(* 2. EMERGENCY STOP LOGIC (Error 12) *)
IF E_Stop_Active THEN
    FOR i := 1 TO 6 DO
        Auto_Bin[i] := FALSE;
        auto_bin_cutoff[i] := FALSE;
        auto_bin_motor[i] := FALSE;
    END_FOR;
    Sequence_Complete := FALSE;
    Active_Material_ID := 0;
    Active_Bin_ID := 0;
    Active_Target_Weight := 0.0;
    Error_Code := 12;
    Status_Message := 'Error 12: Emergency Stop Active!';
    Step := 99;
    Transition_Timer(IN := FALSE);
    Completion_Timer(IN := FALSE);
    RETURN;
END_IF;


(* 3. RECIPE SEQUENCE START *)
IF Step = 0 AND Start_Button THEN
    Step := 1;
    bin_last_weight := load_cell_value;
    Sequence_Complete := FALSE;
    Error_Code := 0;
    Status_Message := 'Auto Batch Started';
    Active_Target_Weight := 0.0;
    (* Clear actual weights and outputs on start *)
    FOR i := 1 TO 6 DO
        Actual_Weights[i] := 0.0;
        Auto_Bin[i] := FALSE;
        auto_bin_cutoff[i] := FALSE;
        auto_bin_motor[i] := FALSE;
    END_FOR;
END_IF;


(* 4. SEQUENCE CONTROL STATE MACHINE *)
CASE Step OF
    0:
        Active_Material_ID := 0;
        Active_Bin_ID := 0;
        Active_Target_Weight := 0.0;
        IF Error_Code = 0 THEN Status_Message := 'Auto Idle'; END_IF;
        
    1..6: (* Discharging Silos 1 to 6 *)
        Mat_Idx := Auto_Bin_Material_Mapping[Step];
        
        IF Mat_Idx = 0 THEN
            (* Skip this bin instantly *)
            Step := Step + 1;
        ELSE
            (* Fetch target weight from global Recipe_Weights array *)
            bin_set_value := GVL.Recipe_Weights[Mat_Idx];
            
            (* Calculate effective target weight (Looked up Target - Tolerance) *)
            target_act_bin := bin_set_value - Auto_Bin_Tolerance[Step];
            Active_Target_Weight := target_act_bin;
            
            (* Calculate weight added by current active bin *)
            actual_bin := load_cell_value - bin_last_weight;
            Actual_Weights[Step] := actual_bin;
            
            (* Calculate cutoff trigger threshold *)
            cutoff_trigger_weight := target_act_bin - Auto_Bin_Cutoff_Weights[Step];
            
            Active_Material_ID := Mat_Idx;
            Active_Bin_ID := Step;
            Status_Message := 'Auto Pouring';
            
            (* COARSE/FINE FEED TRANSITIONS WITH TOLERANCE OFFSETS *)
            IF actual_bin < cutoff_trigger_weight THEN
                (* Phase 1: Coarse Feed (Conveyor Motor ON, Main Valve ON, Fine Cutoff OFF) *)
                Auto_Bin[Step] := TRUE;
                auto_bin_cutoff[Step] := FALSE;
                auto_bin_motor[Step] := TRUE;
            ELSIF actual_bin < target_act_bin THEN
                (* Phase 2: Fine Feed (Conveyor Motor ON, Main Valve OFF, Fine Cutoff ON) *)
                Auto_Bin[Step] := FALSE;
                auto_bin_cutoff[Step] := TRUE;
                auto_bin_motor[Step] := TRUE;
            ELSE
                (* Phase 3: Completed (All OFF) *)
                Auto_Bin[Step] := FALSE;
                auto_bin_cutoff[Step] := FALSE;
                auto_bin_motor[Step] := FALSE;
                bin_last_weight := load_cell_value;
                Active_Target_Weight := 0.0;
                Step := 10 + Step; // Offset to separate transition states
            END_IF;
            
            (* RUNTIME CHECKS *)
            (* Check 21 & 22: Scale Limits *)
            IF load_cell_value > 500.0 THEN
                Error_Code := 21;
                Status_Message := 'Error 21: Scale Overloaded!';
                Step := 99;
                RETURN;
            ELSIF load_cell_value < 0.0 THEN
                Error_Code := 22;
                Status_Message := 'Error 22: Scale Underloaded/Fault!';
                Step := 99;
                RETURN;
            END_IF;
        END_IF;

    11..15: (* Transition Delays (Between Bins) *)
        Active_Material_ID := 0;
        Active_Bin_ID := 0;
        Active_Target_Weight := 0.0;
        Status_Message := 'Transition Delay';
        
        Transition_Timer(IN := TRUE, PT := Step_Delay_Time);
        IF Transition_Timer.Q THEN
            Transition_Timer(IN := FALSE);
            Step := (Step - 10) + 1; // Advance to next bin
        END_IF;
        
    16: (* Transition Delay After Last Bin (Bin 6) Closes *)
        Active_Material_ID := 0;
        Active_Bin_ID := 0;
        Active_Target_Weight := 0.0;
        Status_Message := 'Settling Last Bin';
        
        Transition_Timer(IN := TRUE, PT := Step_Delay_Time);
        IF Transition_Timer.Q THEN
            Transition_Timer(IN := FALSE);
            Step := 7; // Go to post-discharge wait step
        END_IF;

    7: (* Wait 2 Seconds After Closing the Last Bin *)
        Active_Material_ID := 0;
        Active_Bin_ID := 0;
        Active_Target_Weight := 0.0;
        Status_Message := 'Settling Delay';
        Completion_Timer(IN := TRUE, PT := Post_Complete_Delay);
        IF Completion_Timer.Q THEN
            Completion_Timer(IN := FALSE);
            Step := 8; // Proceed to reset last weight
        END_IF;
        
    8: (* Reset bin_last_weight to 0 & Complete *)
        Active_Material_ID := 0;
        Active_Bin_ID := 0;
        Active_Target_Weight := 0.0;
        Status_Message := 'Sequence Completed';
        bin_last_weight := 0.0;
        Sequence_Complete := TRUE;
        
        IF NOT Start_Button THEN
            Step := 0;
            Sequence_Complete := FALSE;
            (* Reset all actual weights at completion once start is released *)
            FOR i := 1 TO 6 DO
                Actual_Weights[i] := 0.0;
            END_FOR;
        END_IF;
        
    99: (* Error Abort state *)
        FOR i := 1 TO 6 DO 
            Auto_Bin[i] := FALSE; 
            auto_bin_cutoff[i] := FALSE;
            auto_bin_motor[i] := FALSE;
        END_FOR;
        Active_Material_ID := 0;
        Active_Bin_ID := 0;
        Active_Target_Weight := 0.0;
        IF NOT Start_Button THEN
            Step := 0;
            Error_Code := 0;
            Status_Message := 'Auto Idle';
        END_IF;
END_CASE;

END_FUNCTION_BLOCK

// PLC_AC500_V3/Application/Manual_Batching_V9
FUNCTION_BLOCK Manual_Batching_V9
VAR_INPUT
    Start_Button : BOOL;      // Signal to start the batching sequence
    E_Stop_Active : BOOL;     // Emergency Stop active signal
    Manual_Bin_Material_Mapping : ARRAY[1..10] OF INT; // Material index mapping for 10 manual silos
    Manual_Bin_Cutoff_Weights : ARRAY[1..10] OF REAL; // Cutoff weight thresholds (kg)
    Manual_Bin_Tolerance : ARRAY[1..10] OF REAL; // Tolerance weight offset values (kg)
END_VAR
VAR_IN_OUT
    load_cell_value : REAL;   // Weight value read/written from load cell
END_VAR
VAR_OUTPUT
    Manual_Bin : ARRAY[1..10] OF BOOL; // Prompts/indicators for Bins 7..16
    manual_bin_cutoff : ARRAY[1..10] OF BOOL; // Manual pre-cutoff indicators
    manual_bin_motor : ARRAY[1..10] OF BOOL; // Main manual feeder motor outputs
    Actual_Weights : ARRAY[1..10] OF REAL; // Actual weight poured per silo
    Sequence_Complete : BOOL;  // Batch complete flag
    Active_Material_ID : INT;  // Currently active ingredient ID
    Active_Bin_ID : INT;       // Currently active physical Bin ID (7..16)
    Active_Target_Weight : REAL; // Recipe target weight of active bin (with tolerance applied)
    Error_Code : INT;          // Active error code
    Status_Message : STRING;   // Diagnostic text message
END_VAR
VAR
    Step : INT := 0;          // State machine index (0: Idle, 1..10: Bins, 11..20: Delays, 30: Settling, 40: Complete, 99: Error)
    bin_last_weight : REAL;   // Baseline weight on the load cell before starting current bin
    actual_bin : REAL;        // Current weight added from active bin
    target_act_bin : REAL;    // Effective target weight to add from the active bin (GVL target - Tolerance)
    bin_set_value : REAL;     // Setpoint weight looked up from GVL
    cutoff_trigger_weight : REAL; // Calculated target threshold weight minus cutoff and tolerance values
    
    Mat_Idx : INT;
    i : INT;                  // General loop index
    
    (* TIMERS FOR TRANSITIONS & DELAYS *)
    Transition_Timer : TON;
    Completion_Timer : TON;
    Step_Delay_Time : TIME := T#2S;
    Post_Complete_Delay : TIME := T#2S;
    
    (* DIAGNOSTIC TIMERS *)
    Operator_Timer : TON;
    
    (* SELF-CONTAINED SIMULATION VARIABLES *)
    Simulation_Mode : BOOL := TRUE;
    Sim_Rate : REAL := 10.0;            // Simulated pouring speed (10.0 kg/s)
    Sim_Timer : TON;
    Start_Sim_Weight : REAL;
    Discharge_Active : BOOL;
END_VAR

(* Manual Batching FB V9 with Tolerance Logic *)

(* 1. SIMULATION WEIGHT MANAGEMENT *)
IF Simulation_Mode AND Step <> 99 THEN
    (* Reset simulation to baseline *)
    IF Step = 0 AND NOT Start_Button AND NOT Sequence_Complete THEN
        load_cell_value := 0.0;
        bin_last_weight := 0.0;
        Start_Sim_Weight := 0.0;
        Sim_Timer(IN := FALSE);
    END_IF;
    
    (* Check if operator is actively pouring *)
    Discharge_Active := FALSE;
    IF Step >= 1 AND Step <= 10 THEN
        Discharge_Active := manual_bin_motor[Step];
    END_IF;
    
    (* Simulate weight gain on the load cell *)
    IF Discharge_Active THEN
        Sim_Timer(IN := TRUE, PT := T#1000S);
        load_cell_value := Start_Sim_Weight + (TIME_TO_REAL(Sim_Timer.ET) / 1000.0) * Sim_Rate;
    ELSE
        Sim_Timer(IN := FALSE);
        Start_Sim_Weight := load_cell_value;
    END_IF;
END_IF;


(* 2. EMERGENCY STOP LOGIC (Error 12) *)
IF E_Stop_Active THEN
    FOR i := 1 TO 10 DO
        Manual_Bin[i] := FALSE;
        manual_bin_cutoff[i] := FALSE;
        manual_bin_motor[i] := FALSE;
    END_FOR;
    Sequence_Complete := FALSE;
    Active_Material_ID := 0;
    Active_Bin_ID := 0;
    Active_Target_Weight := 0.0;
    Error_Code := 12;
    Status_Message := 'Error 12: Emergency Stop Active!';
    Step := 99;
    Transition_Timer(IN := FALSE);
    Completion_Timer(IN := FALSE);
    RETURN;
END_IF;


(* 3. RECIPE SEQUENCE START *)
IF Step = 0 AND Start_Button THEN
    Step := 1;
    bin_last_weight := load_cell_value;
    Sequence_Complete := FALSE;
    Error_Code := 0;
    Status_Message := 'Manual Batch Started';
    Active_Target_Weight := 0.0;
    (* Clear actual weights on start *)
    FOR i := 1 TO 10 DO
        Actual_Weights[i] := 0.0;
        Manual_Bin[i] := FALSE;
        manual_bin_cutoff[i] := FALSE;
        manual_bin_motor[i] := FALSE;
    END_FOR;
END_IF;


(* 4. SEQUENCE CONTROL STATE MACHINE *)
CASE Step OF
    0:
        Active_Material_ID := 0;
        Active_Bin_ID := 0;
        Active_Target_Weight := 0.0;
        IF Error_Code = 0 THEN Status_Message := 'Manual Idle'; END_IF;
        
    1..10: (* Prompts Silos 7 to 16 *)
        Mat_Idx := Manual_Bin_Material_Mapping[Step];
        
        IF Mat_Idx = 0 THEN
            (* Skip this bin instantly *)
            Step := Step + 1;
        ELSE
            (* Fetch target weight from global Recipe_Weights array *)
            bin_set_value := GVL.Recipe_Weights[Mat_Idx];
            
            (* Calculate effective target weight (Looked up Target - Tolerance) *)
            target_act_bin := bin_set_value - Manual_Bin_Tolerance[Step];
            Active_Target_Weight := target_act_bin;
            
            (* Calculate weight added by current active bin *)
            actual_bin := load_cell_value - bin_last_weight;
            Actual_Weights[Step] := actual_bin;
            
            (* Calculate cutoff trigger threshold *)
            cutoff_trigger_weight := target_act_bin - Manual_Bin_Cutoff_Weights[Step];
            
            Active_Material_ID := Mat_Idx;
            Active_Bin_ID := Step + 6;
            Status_Message := 'Manual Pouring Active';
            
            (* COARSE/FINE FEED TRANSITIONS WITH TOLERANCE OFFSETS *)
            IF actual_bin < cutoff_trigger_weight THEN
                (* Phase 1: Coarse Feed (Motor ON, Prompt ON, Cutoff OFF) *)
                Manual_Bin[Step] := TRUE;
                manual_bin_cutoff[Step] := FALSE;
                manual_bin_motor[Step] := TRUE;
            ELSIF actual_bin < target_act_bin THEN
                (* Phase 2: Fine Feed (Motor ON, Prompt OFF, Cutoff ON) *)
                Manual_Bin[Step] := FALSE;
                manual_bin_cutoff[Step] := TRUE;
                manual_bin_motor[Step] := TRUE;
            ELSE
                (* Phase 3: Completed (All OFF) *)
                Manual_Bin[Step] := FALSE;
                manual_bin_cutoff[Step] := FALSE;
                manual_bin_motor[Step] := FALSE;
                bin_last_weight := load_cell_value;
                Active_Target_Weight := 0.0;
                Step := 10 + Step; // Offset to separate transition states
            END_IF;
            
            (* RUNTIME CHECKS *)
            (* Check 21 & 22: Scale Limits *)
            IF load_cell_value > 500.0 THEN
                Error_Code := 21;
                Status_Message := 'Error 21: Scale Overloaded!';
                Step := 99;
                RETURN;
            ELSIF load_cell_value < 0.0 THEN
                Error_Code := 22;
                Status_Message := 'Error 22: Scale Underloaded/Fault!';
                Step := 99;
                RETURN;
            END_IF;
            
            (* Check 30: Operator Timeout *)
            Operator_Timer(IN := manual_bin_motor[Step], PT := T#300S);
            IF Operator_Timer.Q THEN
                Error_Code := 30;
                Status_Message := 'Error 30: Manual Operator Timeout!';
                Step := 99;
                RETURN;
            END_IF;
        END_IF;

    11..19: (* Transition Delays (Between Bins) *)
        Active_Material_ID := 0;
        Active_Bin_ID := 0;
        Active_Target_Weight := 0.0;
        Status_Message := 'Transition Delay';
        Transition_Timer(IN := TRUE, PT := Step_Delay_Time);
        IF Transition_Timer.Q THEN
            Transition_Timer(IN := FALSE);
            Step := (Step - 10) + 1; // Advance to next bin
        END_IF;
        
    20: (* Transition Delay After Last Bin (Bin 10) Closes *)
        Active_Material_ID := 0;
        Active_Bin_ID := 0;
        Active_Target_Weight := 0.0;
        Status_Message := 'Settling Last Bin';
        Transition_Timer(IN := TRUE, PT := Step_Delay_Time);
        IF Transition_Timer.Q THEN
            Transition_Timer(IN := FALSE);
            Step := 30; // Go to post-discharge wait step (State 30)
        END_IF;

    30: (* Wait 2 Seconds After Closing the Last Bin *)
        Active_Material_ID := 0;
        Active_Bin_ID := 0;
        Active_Target_Weight := 0.0;
        Status_Message := 'Settling Delay';
        Completion_Timer(IN := TRUE, PT := Post_Complete_Delay);
        IF Completion_Timer.Q THEN
            Completion_Timer(IN := FALSE);
            Step := 40; // Proceed to reset last weight (State 40)
        END_IF;
        
    40: (* Reset bin_last_weight to 0 & Complete *)
        Active_Material_ID := 0;
        Active_Bin_ID := 0;
        Active_Target_Weight := 0.0;
        Status_Message := 'Sequence Completed';
        bin_last_weight := 0.0;
        Sequence_Complete := TRUE;
        
        IF NOT Start_Button THEN
            Step := 0;
            Sequence_Complete := FALSE;
            (* Reset all actual weights at completion once start is released *)
            FOR i := 1 TO 10 DO
                Actual_Weights[i] := 0.0;
            END_FOR;
        END_IF;
        
    99: (* Error Abort state *)
        FOR i := 1 TO 10 DO 
            Manual_Bin[i] := FALSE;
            manual_bin_cutoff[i] := FALSE;
            manual_bin_motor[i] := FALSE;
        END_FOR;
        Active_Material_ID := 0;
        Active_Bin_ID := 0;
        Active_Target_Weight := 0.0;
        IF NOT Start_Button THEN
            Step := 0;
            Error_Code := 0;
            Status_Message := 'Manual Idle';
        END_IF;
END_CASE;

END_FUNCTION_BLOCK

// PLC_AC500_V3/Application/batching9
PROGRAM batching9
VAR
    Auto_Ctrl : Auto_Batching_V9;
    Manual_Ctrl : Manual_Batching_V9;
    
    (* Global Inputs & Toggles *)
    Start_Button : BOOL;
    E_Stop_Active : BOOL;
    
    (* Parallel Weight Feedbacks *)
    load_cell_auto : REAL;
    load_cell_manual : REAL;
    
    (* Sub-Block Diagnostic Indicators - Ordered exactly below loadcell *)
    Auto_Active_Mat : INT;
    Auto_Active_Bin : INT;
    Auto_Active_Target : REAL; // Active Target Weight for Auto (displays GVL setpoint - Tolerance)
    Auto_Err : INT;
    Auto_Msg : STRING;
    
    Manual_Active_Mat : INT;
    Manual_Active_Bin : INT;
    Manual_Active_Target : REAL; // Active Target Weight for Manual (displays GVL setpoint - Tolerance)
    Manual_Err : INT;
    Manual_Msg : STRING;
    
    (* Process Outputs *)
    Auto_Bin : ARRAY[1..6] OF BOOL; // Valve control outputs (Coarse)
    auto_bin_cutoff : ARRAY[1..6] OF BOOL; // Cutoff indicators (Fine)
    auto_bin_motor : ARRAY[1..6] OF BOOL; // Conveyor/feeder motor outputs
    
    Manual_Bin : ARRAY[1..10] OF BOOL; // Prompt indicators (Coarse)
    manual_bin_cutoff : ARRAY[1..10] OF BOOL; // Cutoff indicators (Fine)
    manual_bin_motor : ARRAY[1..10] OF BOOL; // Conveyor/feeder motor outputs
    
    Auto_Weights : ARRAY[1..6] OF REAL;
    Manual_Weights : ARRAY[1..10] OF REAL;
    
    Auto_Complete : BOOL;
    Manual_Complete : BOOL;
    Sequence_Complete : BOOL;
    
    (* Diagnostics & Interlocks *)
    Error_Code : INT := 0;
    Status_Message : STRING := 'System Ready';
    
    (* Array Configurations & Mapping - Renamed for clarity *)
    Auto_Bin_Material_Mapping : ARRAY[1..6] OF INT := [1, 2, 0, 4, 5, 6];
    Manual_Bin_Material_Mapping : ARRAY[1..10] OF INT := [7, 8, 0, 10, 11, 12, 13, 14, 15, 16];
    Auto_Bin_Cutoff_Weights : ARRAY[1..6] OF REAL := [2.0, 1.5, 0.0, 3.0, 5.0, 1.0]; // Cutoff margins (kg)
    Manual_Bin_Cutoff_Weights : ARRAY[1..10] OF REAL := [2.0, 1.5, 0.0, 3.0, 5.0, 1.0, 2.0, 2.0, 2.0, 2.0];
    Auto_Bin_Tolerance : ARRAY[1..6] OF REAL := [1.0, 0.5, 0.0, 1.0, 2.0, 0.5]; // Tolerance offsets (kg)
    Manual_Bin_Tolerance : ARRAY[1..10] OF REAL := [1.0, 0.5, 0.0, 1.0, 2.0, 0.5, 1.0, 1.0, 1.0, 1.0];
    
    i : INT;
    j : INT;
    Duplicate_Found : BOOL;
    Invalid_Material_Range : BOOL;
    Zero_Target_Found : BOOL;
    Conf_Err_Id : INT;
END_VAR

(* 1. STARTUP CONFIGURATION CHECKS *)
Duplicate_Found := FALSE;
Invalid_Material_Range := FALSE;
Zero_Target_Found := FALSE;

FOR i := 1 TO 6 DO
    (* Check 2: Out of Range (Auto) *)
    IF Auto_Bin_Material_Mapping[i] < 0 OR Auto_Bin_Material_Mapping[i] > 20 THEN
        Invalid_Material_Range := TRUE;
    END_IF;
    
    (* Check 3: Zero Target (Auto) *)
    IF Auto_Bin_Material_Mapping[i] <> 0 AND Auto_Bin_Material_Mapping[i] <= 20 THEN
        IF GVL.Recipe_Weights[Auto_Bin_Material_Mapping[i]] = 0.0 THEN
            Zero_Target_Found := TRUE;
        END_IF;
    END_IF;
    
    (* Check 1: Duplicate Cross-Array Material ID *)
    IF Auto_Bin_Material_Mapping[i] <> 0 AND Auto_Bin_Material_Mapping[i] <= 20 THEN
        FOR j := 1 TO 10 DO
            IF Auto_Bin_Material_Mapping[i] = Manual_Bin_Material_Mapping[j] THEN
                Duplicate_Found := TRUE;
            END_IF;
        END_FOR;
    END_IF;
END_FOR;

FOR j := 1 TO 10 DO
    (* Check 2: Out of Range (Manual) *)
    IF Manual_Bin_Material_Mapping[j] < 0 OR Manual_Bin_Material_Mapping[j] > 20 THEN
        Invalid_Material_Range := TRUE;
    END_IF;
    
    (* Check 3: Zero Target (Manual) *)
    IF Manual_Bin_Material_Mapping[j] <> 0 AND Manual_Bin_Material_Mapping[j] <= 20 THEN
        IF GVL.Recipe_Weights[Manual_Bin_Material_Mapping[j]] = 0.0 THEN
            Zero_Target_Found := TRUE;
        END_IF;
    END_IF;
END_FOR;

(* Configuration Error Resolution *)
IF Duplicate_Found THEN
    Error_Code := 1;
    Status_Message := 'Error 1: Duplicate Material ID mapped in Auto and Manual!';
ELSIF Invalid_Material_Range THEN
    Error_Code := 2;
    Status_Message := 'Error 2: Material Index configuration out of range (1..20)!';
ELSIF Zero_Target_Found THEN
    Error_Code := 3;
    Status_Message := 'Error 3: Configured Material ID has a 0.0 kg target weight!';
ELSE
    IF Error_Code <= 3 THEN
        Error_Code := 0;
    END_IF;
END_IF;

(* Abort sequences if a configuration error exists *)
IF Error_Code >= 1 AND Error_Code <= 3 THEN
    FOR i := 1 TO 6 DO Auto_Bin[i] := FALSE; auto_bin_cutoff[i] := FALSE; auto_bin_motor[i] := FALSE; END_FOR;
    FOR i := 1 TO 10 DO Manual_Bin[i] := FALSE; manual_bin_cutoff[i] := FALSE; manual_bin_motor[i] := FALSE; END_FOR;
    Auto_Ctrl(Start_Button := FALSE, E_Stop_Active := TRUE, load_cell_value := load_cell_auto);
    Manual_Ctrl(Start_Button := FALSE, E_Stop_Active := TRUE, load_cell_value := load_cell_manual);
    Auto_Active_Target := 0.0;
    Manual_Active_Target := 0.0;
    RETURN;
END_IF;


(* 2. CONCURRENT EXECUTION OF FB INSTANCES *)
Auto_Ctrl(
    Start_Button := Start_Button,
    E_Stop_Active := E_Stop_Active,
    load_cell_value := load_cell_auto,
    Auto_Bin_Material_Mapping := Auto_Bin_Material_Mapping,
    Auto_Bin_Cutoff_Weights := Auto_Bin_Cutoff_Weights,
    Auto_Bin_Tolerance := Auto_Bin_Tolerance,
    Auto_Bin => Auto_Bin,
    auto_bin_cutoff => auto_bin_cutoff,
    auto_bin_motor => auto_bin_motor,
    Actual_Weights => Auto_Weights,
    Sequence_Complete => Auto_Complete,
    Active_Material_ID => Auto_Active_Mat,
    Active_Bin_ID => Auto_Active_Bin,
    Active_Target_Weight => Auto_Active_Target,
    Error_Code => Auto_Err,
    Status_Message => Auto_Msg
);

Manual_Ctrl(
    Start_Button := Start_Button,
    E_Stop_Active := E_Stop_Active,
    load_cell_value := load_cell_manual,
    Manual_Bin_Material_Mapping := Manual_Bin_Material_Mapping,
    Manual_Bin_Cutoff_Weights := Manual_Bin_Cutoff_Weights,
    Manual_Bin_Tolerance := Manual_Bin_Tolerance,
    Manual_Bin => Manual_Bin,
    manual_bin_cutoff => manual_bin_cutoff,
    manual_bin_motor => manual_bin_motor,
    Actual_Weights => Manual_Weights,
    Sequence_Complete => Manual_Complete,
    Active_Material_ID => Manual_Active_Mat,
    Active_Bin_ID => Manual_Active_Bin,
    Active_Target_Weight => Manual_Active_Target,
    Error_Code => Manual_Err,
    Status_Message => Manual_Msg
);

(* Runtime Error Mapping & Aggregation *)
IF Auto_Err <> 0 THEN
    Error_Code := Auto_Err;
    Status_Message := CONCAT('Auto Error: ', Auto_Msg);
ELSIF Manual_Err <> 0 THEN
    Error_Code := Manual_Err;
    Status_Message := CONCAT('Manual Error: ', Manual_Msg);
ELSE
    Error_Code := 0;
    
    Sequence_Complete := Auto_Complete AND Manual_Complete;
    IF Sequence_Complete THEN
        Status_Message := 'Batch Sequence Completed';
    ELSIF Start_Button THEN
        Status_Message := 'Batch Sequence Running';
    ELSE
        Status_Message := 'System Ready';
    END_IF;
END_IF;

END_PROGRAM

// PLC_AC500_V3/Application/batching4_vis
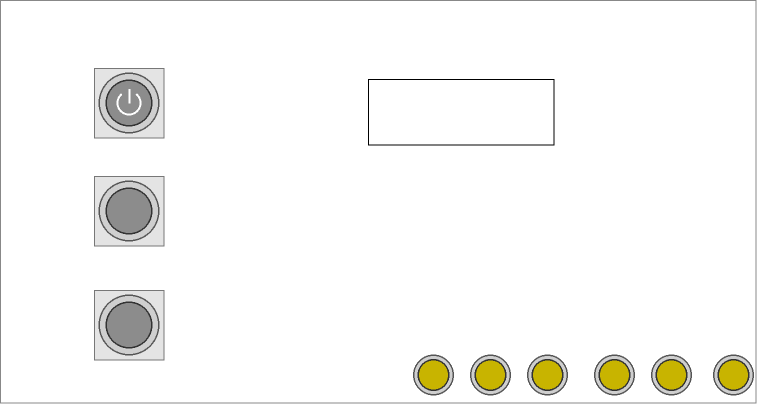
VISUALIZATION batching4_vis  // 757x404
    PushSwitch (94,290 70x70), behaviour: TOGGLE, style: Switch-PushSwitch-Gray
    PushSwitch (94,176 70x70), behaviour: TOGGLE, style: Switch-PushSwitch-Gray
    PowerSwitch (94,68 70x70), behaviour: TOGGLE, style: Switch-PowerSwitch-Gray
    Lamp1 (591,346 47x58), style: Lamp-Lamp1-Yellow
    Lamp1 (524,346 47x58), style: Lamp-Lamp1-Yellow
    Lamp1 (467,346 47x58), style: Lamp-Lamp1-Yellow
    Lamp1 (410,346 47x58), style: Lamp-Lamp1-Yellow
    Lamp1 (648,346 47x58), style: Lamp-Lamp1-Yellow
    Lamp1 (710,346 47x58), style: Lamp-Lamp1-Yellow
    Rectangle (368,79 186x66)
END_VISUALIZATION

(* text list Diag_IO_Bus (id | default | en | de | fr | es | zh)
  Err_1037 | Test error | Test error | Testfehler |  |  | 测试错误
  Err_12 | Test pulse error -> Check wiring and sensor | Test pulse error -> Check wiring and sensor | Testimpuls-Fehler -> Verdrahtung und Sensor prüfen |  |  | 测试脉冲错误 -> 检查接线和传感器
  Err_13 | Test pulse cross-talk error -> Check wiring and sensor. If this error persists, replace I/O module. Contact ABB technical support. | Test pulse cross-talk error -> Check wiring and sensor. If this error persists, replace I/O module. Contact ABB technical support. | Fehler Testimpuls Kanalübersprechen  -> Verdrahtung und Sensor prüfen. Falls der Fehler weiterhin besteht, E/A-Modul austauschen. Technischen Support von ABB kontaktieren. |  |  | 测试脉冲串扰错误 -> 检查接线和传感器. 如果此错误仍然存在，请更换 I/O 模块. 联系 ABB 技术支持.
  Err_16128 | Failed max wait run | Failed max wait run | Lauf max. Warten fehlgeschlagen |  |  | 最大等待运行失败
  Err_16129 | Critical error, see log | Critical error, see log | Kritischer Fehler, siehe Protokoll |  |  | 严重错误，请参阅日志
  Err_16130 | Fatal error, see log | Fatal error, see log | Schwerwiegender Fehler, siehe Protokoll |  |  | 致命错误，请参阅日志
  Err_16131 | Timeout -> Replace I/O module | Timeout -> Replace I/O module | Timeout -> E/A-Modul austauschen |  |  | 超时 -> 更换 I/O 模块
  Err_16133 | Output data size mismatch | Output data size mismatch | Diskrepanz Ausgangsdatengröße |  |  | 输出数据大小不匹配
  Err_16134 | Input data size mismatch | Input data size mismatch | Diskrepanz Eingangsdatengröße |  |  | 输入数据大小不匹配
  Err_16137 | Overflow diagnosis buffer -> Restart | Overflow diagnosis buffer -> Restart | Überlauf Diagnosepuffer -> Neu Starten |  |  | 诊断缓冲区溢出 -> 重新启动
  Err_16138 | Non-safety I/O: Voltage overflow at outputs (above UP3 level), Safety I/O: Process voltage too high -> Check terminals / Check process voltage | Non-safety I/O: Voltage overflow at outputs (above UP3 level), Safety I/O: Process voltage too high -> Check terminals / Check process voltage | Standard-E/A: Spannungsüberlauf an Ausgängen (über UP3-Niveau), Sicherheits-E/A: Prozessspannung zu hoch -> Terminals prüfen / Prozessspannung prüfen |  |  | 非安全 I/O：输出端电压溢出（高于 UP3 电平），安全 I/O：过程电压过高 -> 检查终端 / 检查过程电压
  Err_16139 | Process voltage UP or UP3 too low -> Check process voltage | Process voltage UP or UP3 too low -> Check process voltage | Prozessspannung UP oder UP3 zu niedrig -> Prozessspannung prüfen |  |  | 过程电压 UP 或 UP3 过低 -> 检查过程电压
  Err_16145 | Error setting parameters | Error setting parameters | Fehlereinstellungsparameter |  |  | 设置参数时出错
  Err_16146 | Plausibility check failed (iParameter) -> Check configuration | Plausibility check failed (iParameter) -> Check configuration | Plausibilitätsprüfung fehlgeschlagen (iParameter) -> Konfiguration überprüfen |  |  | 合理性检查失败（i 参数） -> 检查配置
  Err_16147 | Checksum error -> Non-safety I/O: Replace I/O module. Safety I/O: Check safety configuration and CRCs for I- and F-Parameters. | Checksum error -> Non-safety I/O: Replace I/O module. Safety I/O: Check safety configuration and CRCs for I- and F-Parameters. | Prüfsummenfehler -> Standard-E/A: E/A-Modul austauschen. Sicherheits-E/A: Sicherheitskonfiguration und CRCs auf I- und F-Parameter prüfen. |  |  | 检校验和错误 -> 非安全 I/O：更换 I/O 模块. 安全 I/O：检查 I 参数和 F 参数的安全配置和 CRC.
  Err_16148 | PROFIsafe communication error -> Restart I/O module. If this error persists, contact ABB technical support. | PROFIsafe communication error -> Restart I/O module. If this error persists, contact ABB technical support. | PROFIsafe-Kommunikationsfehler -> E/A-Modul neu starten. Falls der Fehler weiterhin besteht, technischen Support von ABB kontaktieren. |  |  | PROFIsafe 通信错误 -> 重新启动 I/O 模块. 如果此错误仍然存在，请联系 ABB 技术支持.
  Err_16149 | No module data | No module data | Keine Moduldaten |  |  | 无模块数据
  Err_16153 | PROFIsafe watchdog timed out -> Restart I/O module. If this error persists, increase PROFIsafe watchdog time. | PROFIsafe watchdog timed out -> Restart I/O module. If this error persists, increase PROFIsafe watchdog time. | Timeout von PROFIsafe-Watchdog -> E/A-Modul neu starten. Falls der Fehler weiterhin besteht, PROFIsafe-Watchdog-Zeit verlängern. |  |  | PROFIsafe 看门狗超时 -> 重新启动 I/O 模块. 如果此错误仍然存在，请增加 PROFIsafe 看门狗时间.
  Err_16154 | Size of parameters expected by module differs from size provided by configuration -> Check master or configuration | Size of parameters expected by module differs from size provided by configuration -> Check master or configuration | Vom Modul erwartete Parametergröße weicht von der in der Konfiguration angegebenen Größe ab -> Master oder Konfiguration überprüfen |  |  | 模块期望的参数大小与配置提供的参数大小不同 -> 检查主设备或配置
  Err_16156 | F-Parameter configuration and address switch value do not match -> Check I/O module F-Parameter configuration and module address switch value. | F-Parameter configuration and address switch value do not match -> Check I/O module F-Parameter configuration and module address switch value. | Konfiguration für F-Parameter und Wert des Adressschalters stimmen nicht überein -> Konfiguration für F-Parameter des E/A-Moduls und Wert des Adressschalters überprüfen. |  |  | F 参数配置和地址开关值不匹配 -> 检查 I/O 模块 F 参数配置和模块地址开关值.
  Err_16158 | Type of present module does not match configuration | Type of present module does not match configuration | Typ des vorhandenen Moduls stimmt nicht mit Konfiguration überein |  |  | 当前模块类型与配置不匹配
  Err_16159 | Configured number of modules differs from found ones | Configured number of modules differs from found ones | Konfigurierte Anzahl von Modulen weicht von Anzahl gefundener Module ab |  |  | 配置的模块数量与找到的模块数量不同
  Err_16160 | At least one module failed during configuration | At least one module failed during configuration | Mindestens ein Modul während Konfiguration ausgefallen |  |  | 配置期间至少有一个模块发生故障
  Err_16164 | Internal data exchange failure -> Replace I/O module | Internal data exchange failure -> Replace I/O module | Fehler interner Datenaustausch -> E/A-Modul austauschen |  |  | 内部数据交换失败 -> 更换 I/O 模块
  Err_16168 | Different hard-/firmware versions in the module -> Replace I/O module | Different hard-/firmware versions in the module -> Replace I/O module | Unterschiedliche Hardware-/Firmware-Versionen im Modul -> E/A-Modul austauschen |  |  | 模块中的硬件/固件版本不同 -> 更换 I/O 模块
  Err_16171 | Internal error -> Replace I/O module | Internal error -> Replace I/O module | Interner Fehler -> E/A-Modul austauschen |  |  | 内部错误 -> 更换 I/O 模块
  Err_16172 | Has not passed factory test | Has not passed factory test | Hat Werksprüfung nicht bestanden |  |  | 未通过出厂测试
  Err_16173 | No process voltage UP or UP3 -> Check process voltage | No process voltage UP or UP3 -> Check process voltage | Keine Prozessspannung UP oder UP3 -> Prozessspannung prüfen |  |  | 无过程电压 UP 或 UP3 -> 检查过程电压
  Err_16175 | Sensor voltage too low | Sensor voltage too low | Sensorspannung zu niedrig |  |  | 传感器电压过低
  Err_16194 | Fatal error, not running any more | Fatal error, not running any more | Schwerwiegender Fehler, Ausführung gestoppt |  |  | 致命错误，不再运行
  Err_16246 | Failed to start the parameterization of modules | Failed to start the parameterization of modules | Starten von Parametrierung für Module fehlgeschlagen |  |  | 无法启动模块的参数化
  Err_16247 | Failed setting parameters | Failed setting parameters | Einstellen von Parametern fehlgeschlagen |  |  | 设置参数失败
  Err_16248 | Failed setting expected module | Failed setting expected module | Einstellen des erwarteten Moduls fehlgeschlagen |  |  | 设置预期模块失败
  Err_16254 | Size of parameters expected by module differs from size provided by configuration | Size of parameters expected by module differs from size provided by configuration | Vom Modul erwartete Parametergröße weicht von der in der Konfiguration angegebenen Größe ab |  |  | 模块期望的参数大小与配置提供的参数大小不同
  Err_18 | Test error | Test error | Testfehler |  |  | 测试错误
  Err_25 | Stuck at error -> Check I/O module wiring. Restart I/O module, if needed. If this error persists, replace I/O module. | Stuck at error -> Check I/O module wiring. Restart I/O module, if needed. If this error persists, replace I/O module. | Hängengeblieben bei Fehler -> Verdrahtung des E/A-Moduls überprüfen. Bei Bedarf E/A-Modul neu starten. Falls der Fehler weiterhin besteht, E/A-Modul austauschen. |  |  | 卡在错误处 -> 检查 I/O 模块接线. 如果需要，重新启动 I/O 模块. 如果此错误仍然存在，请更换 I/O 模块.
  Err_257 | Wrong measurement, false temperature at the compensation channel | Wrong measurement, false temperature at the compensation channel | Falscher Messwert, falsche Temperatur an Kompensationskanal |  |  | 测量值错误，补偿通道温度错误
  Err_258 | AI531: Wrong measurement; potential difference is too high; CD522: PWM duty cycle out of duty area | AI531: Wrong measurement; potential difference is too high; CD522: PWM duty cycle out of duty area | AI531: Falscher Messwert; Potenzialdifferenz zu hoch; CD522: PWM-Einschaltdauer außerhalb des Einschaltbereichs |  |  | AI531：测量错误; 电位差过高; CD522: PWM 占空比超出占空比范围
  Err_260 | Measurement overflow -> Check channel wiring and sensor power supply | Measurement overflow -> Check channel wiring and sensor power supply | Messwertüberschreitung -> Kanalverdrahtung und Spannungsversorgung des Sensors prüfen |  |  | 测量值溢出 -> 检查通道接线和传感器电源
  Err_263 | Measurement underflow -> Check channel wiring and sensor power supply | Measurement underflow -> Check channel wiring and sensor power supply | Messwertunterschreitung -> Kanalverdrahtung und Spannungsversorgung des Sensors prüfen |  |  | 测量值下溢 -> 检查通道接线和传感器电源
  Err_266 | Short circuit and cut wire or "out of range" | Short circuit and cut wire or "out of range" | Kurzschluss und Drahtbruch oder „außerhalb des zulässigen Bereichs“ |  |  | 短路和断线或“超出范围”
  Err_267 | Output/process voltage too low | Output/process voltage too low | Ausgangs-/Prozessspannung zu gering |  |  | 输出/过程电压过低
  Err_273 | Test error | Test error | Testfehler |  |  | 测试错误
  Err_28 | Cross-talk error -> Check I/O module wiring. Restart I/O module, if needed. If this error persists, replace I/O module. | Cross-talk error -> Check I/O module wiring. Restart I/O module, if needed. If this error persists, replace I/O module. | Fehler Kanalübersprechen -> Verdrahtung des E/A-Moduls überprüfen. Bei Bedarf E/A-Modul neu starten. Falls der Fehler weiterhin besteht, E/A-Modul austauschen. |  |  | 串扰错误 -> 检查 I/O 模块接线. 如果需要，重新启动 I/O 模块. 如果此错误仍然存在，请更换 I/O 模块.
  Err_3 | Discrepancy time expired -> Check discrepancy time value, channel wiring and sensor. | Discrepancy time expired -> Check discrepancy time value, channel wiring and sensor. | Diskrepanzzeit abgelaufen -> Diskrepanzzeit-Wert, Kanalverdrahtung und Sensor überprüfen. |  |  | 偏差时间已过 -> 检查差异时间值、通道接线和传感器.
  Err_303 | Short circuit at analog input -> Check channel wiring | Short circuit at analog input -> Check channel wiring | Kurzschluss an Analogeingang -> Kanalverdrahtung prüfen |  |  | 模拟输入端短路 -> 检查通道接线
  Err_304 | Analog value overflow or broken wire at an analog input -> Check value or check terminals | Analog value overflow or broken wire at an analog input -> Check value or check terminals | Analogwert-Überlauf oder Drahtbruch an Analogeingang -> Wert oder Terminals prüfen |  |  | 模拟输入端模拟值溢出或断线 -> 检查值或检查终端
  Err_311 | Value difference too high -> Adjust tolerance window for channels. Check channel wiring and sensor configuration. | Value difference too high -> Adjust tolerance window for channels. Check channel wiring and sensor configuration. | Wertdifferenz zu groß -> Toleranzfenster für Kanäle einstellen. Kanalverdrahtung und Sensorkonfiguration prüfen. |  |  | 值差异过大 -> 调整通道的容差范围. 检查通道接线和传感器配置.
  Err_524 | Stuck at error | Stuck at error | Hängengeblieben bei Fehler |  |  | 卡在错误处
  Err_525 | Readback error -> Check I/O module wiring. Restart I/O module, if needed. If this error persists, replace I/O module. | Readback error -> Check I/O module wiring. Restart I/O module, if needed. If this error persists, replace I/O module. | Fehler Rücklesen -> Verdrahtung des E/A-Moduls überprüfen. Bei Bedarf E/A-Modul neu starten. Falls der Fehler weiterhin besteht, E/A-Modul austauschen. |  |  | 回读错误 -> 检查 I/O 模块接线. 如果需要，重新启动 I/O 模块. 如果此错误仍然存在，请更换 I/O 模块.
  Err_530 | Class 3: Cross-talk error; Class 4: Internal fuse at 0V is defect. 0V not connected with GND -> Check I/O module wiring. Restart I/O module, if needed. If this error persists, replace I/O module. | Class 3: Cross-talk error; Class 4: Internal fuse at 0V is defect. 0V not connected with GND -> Check I/O module wiring. Restart I/O module, if needed. If this error persists, replace I/O module. | Klasse 3: Fehler Kanalübersprechen; Klasse 4: Interne Sicherung an 0 V defekt. 0 V nicht an GND angeschlossen -> Verdrahtung des E/A-Moduls überprüfen. Bei Bedarf E/A-Modul neu starten. Falls der Fehler weiterhin besteht, E/A-Modul austauschen. |  |  | 3 级：串扰错误; 4 级：0V 时内部保险丝有缺陷. 0V 未连接 GND -> 检查 I/O 模块接线. 如果需要，重新启动 I/O 模块. 如果此错误仍然存在，请更换 I/O 模块.
  Err_540 | Test error | Test error | Testfehler |  |  | 测试错误
  Err_555 | Internal error | Internal error | Interner Fehler |  |  | 内部错误
  Err_559 | Short circuit at digital output -> Check channel wiring | Short circuit at digital output -> Check channel wiring | Kurzschluss an Digitalausgang -> Kanalverdrahtung prüfen |  |  | 数字输出端短路 -> 检查通道接线
  Err_772 | Measurement overflow -> Check channel wiring | Measurement overflow -> Check channel wiring | Messwertüberschreitung -> Kanalverdrahtung prüfen |  |  | 测量值溢出 -> 检查通道接线
  Err_775 | Measurement underflow at analog input -> Check channel wiring | Measurement underflow at analog input -> Check channel wiring | Messwertunterschreitung an Analogausgang -> Kanalverdrahtung prüfen |  |  | 模拟输入端测量值下溢 -> 检查通道接线
  Err_796 | Different configuration | Different configuration | Abweichende Konfiguration |  |  | 配置不同
  Err_8480 | Not supported protocol variant | Not supported protocol variant | Nicht unterstützte Protokollvariante |  |  | 不支持的协议变体
  Err_8482 | Class 2: Timeout while initializing; Class 4: Timeout while waiting for ready status | Class 2: Timeout while initializing; Class 4: Timeout while waiting for ready status | Klasse 2: Timeout bei Initialisierung; Klasse 4: Timeout beim Warten auf Status „Bereit“ |  |  | 2 级：初始化超时; 4 级：等待就绪状态超时
  Err_8483 | Timeout during parameterization | Timeout during parameterization | Timeout bei Parametrierung |  |  | 参数化期间超时
  Err_8707 | PROFIsafe watchdog timed out | PROFIsafe watchdog timed out | Timeout von PROFIsafe-Watchdog |  |  | PROFIsafe 看门狗超时
  Err_8708 | Overvoltage | Overvoltage | Überspannung |  |  | 过电压
  Err_8711 | Undervoltage | Undervoltage | Unterspannung |  |  | 欠电压
  Err_8722 | Internal error | Internal error | Interner Fehler |  |  | 内部错误
  Err_8723 | Checksum error has occured in iParameters | Checksum error has occured in iParameters | Prüfsummenfehler in iParameter |  |  | i 参数中出现校验和错误
  Err_8724 | PROFIsafe communication error | PROFIsafe communication error | PROFIsafe-Kommunikationsfehler |  |  | PROFIsafe 通信错误
  Err_8732 | Internal error | Internal error | Interner Fehler |  |  | 内部错误
  Err_8747 | Internal runtime error | Internal runtime error | Interner Laufzeitfehler |  |  | 内部运行时错误
  Err_8961 | Wrong parameter value, check configuration | Wrong parameter value, check configuration | Falscher Parameterwert, Konfiguration prüfen |  |  | 参数值错误，请检查配置
  Err_8979 | Checksum error has occured in iParameter or F-Parameters | Checksum error has occured in iParameter or F-Parameters | Prüfsummenfehler in iParameter oder F-Parametern |  |  | i 参数或 F 参数中出现校验和错误
  Err_8986 | Invalid configuration -> Check modules and parameterization | Invalid configuration -> Check modules and parameterization | Ungültige Konfiguration -> Module und Parametrierung prüfen |  |  | 配置无效 -> 检查模块和参数化
  Err_8988 | F-Parameter configuration and address switch value do not match -> Check I/O module F-Parameter configuration and module address switch value. | F-Parameter configuration and address switch value do not match -> Check I/O module F-Parameter configuration and module address switch value. | Konfiguration für F-Parameter und Wert des Adressschalters stimmen nicht überein -> Konfiguration für F-Parameter des E/A-Moduls und Wert des Adressschalters überprüfen. |  |  | F 参数配置和地址开关值不匹配 -> 检查 I/O 模块 F 参数配置和模块地址开关值.
  Err_9249 | Timeout while waiting for Reset | Timeout while waiting for Reset | Timeout beim Warten auf Zurücksetzen |  |  | 等待重置时超时
  Err_9258 | Breakdown, communication lost | Breakdown, communication lost | Ausfall, Kommunikation unterbrochen |  |  | 故障，通信中断
  Err_9480 | I/O module removed from hotswap terminal unit or defective module on hotswap terminal unit -> Plug I/O module, replace I/O module | I/O module removed from hotswap terminal unit or defective module on hotswap terminal unit -> Plug I/O module, replace I/O module | E/A-Modul von Hotswap-Terminal-Einheit entfernt oder defektes Modul an Hotswap-Terminal-Einheit -> E/A-Modul einstecken, E/A-Modul austauschen |  |  | I/O 模块已从热插拔终端单元上拔下，或热插拔终端单元上的模块有故障 -> 插入 I/O 模块，更换 I/O 模块
  Err_9500 | Wrong I/O module plugged on hotswap terminal unit -> Remove wrong I/O module and plug projected I/O module | Wrong I/O module plugged on hotswap terminal unit -> Remove wrong I/O module and plug projected I/O module | Falsches E/A-Modul an Hotwwap-Terminal-Einheit eingesteckt -> Falsches E/A-Modul entfernen oder projektiertes E/A-Modul einstecken |  |  | 热插拔终端单元上插入了错误的 I/O 模块 -> 拔出错误的 I/O 模块并插入预计的 I/O 模块
  Err_9514 | No communication with I/O module on hotswap terminal unit -> Replace I/O module | No communication with I/O module on hotswap terminal unit -> Replace I/O module | Keine Kommunikation mit E/A-Modul an Hotswap-Terminal-Einheit -> E/A-Modul austauschen |  |  | 无法与热插拔终端单元上的 I/O 模块通信 -> 更换 I/O 模块
  Err_9526 | I/O module does not support hotswap functionality -> Power off system and replace I/O module | I/O module does not support hotswap functionality -> Power off system and replace I/O module | E/A-Modul unterstützt keine Hotswap-Funktion -> System abschalten und E/A-Modul austauschen |  |  | I/O 模块不支持热插拔功能 -> 关闭系统电源并更换 I/O 模块
  Err_9736 | hotswap terminal unit required but not found | hotswap terminal unit required but not found | Hotswap-Terminal-Einheit erforderlich, jedoch nicht gefunden |  |  | 需要热插拔终端单元但未找到
  Err_9764 | Defective hotswap terminal unit | Defective hotswap terminal unit | Defekte Hotswap-Terminal-Einheit |  |  | 热插拔终端单元有缺陷
  Err_9770 | No communication with hotswap terminal unit -> Restart, if error persists replace terminal unit | No communication with hotswap terminal unit -> Restart, if error persists replace terminal unit | Keine Kommunikation mit Hotswap-Terminal-Einheit -> Neu starten, falls Fehler weiterhin besteht, Terminal-Einheit austauschen |  |  | 无法与热插拔终端单元通信 -> 重新启动，如果错误仍然存在，请更换终端单元
  Hwd_14 | I/O bus | I/O bus | E/A-Bus |  |  | I/O 总线
  Sub1_ | Module | Module | Modul |  |  | 模块
  Sub2_ | Channel | Channel | Kanal |  |  | 通道 *)

(* text list Diag_V3_PLC (id | default | en | de | fr | es | zh)
  Add_570425344 | Unknown reason | Unknown reason | Unbekannter Fehler |  |  | 未知原因
  Add_570425345 | Shutdown of the PLC | Shutdown of the PLC | Abschaltung der SPS |  |  | 关闭 PLC
  Add_570425346 | Reset after having stopped the IEC application | Reset after having stopped the IEC application | Nach Stoppen der IEC-Anwendung zurücksetzen |  |  | 在停止 IEC 应用程序后重置
  Add_570425347 | Exception occurred | Exception occurred | Ausnahme aufgetreten |  |  | 发生异常
  Add_570425348 | IEC application stopped by user | IEC application stopped by user | IEC-Anwendung durch Benutzer gestoppt |  |  | IEC 应用程序由用户停止
  Add_570425349 | IEC application stopped by function block | IEC application stopped by function block | IEC-Anwendung durch Funktionsbaustein gestoppt |  |  | IEC 应用程序由功能块停止
  Add_570425350 | IEC application will be deleted after the stop | IEC application will be deleted after the stop | IEC-Anwendung wird nach Stopp gelöscht |  |  | IEC 应用程序将在停止后被删除
  Add_570425351 | IEC application stopped because of debugging | IEC application stopped because of debugging | IEC-Anwendung wegen Debugging gestoppt |  |  | IEC 应用程序因调试而停止
  Add_570425352 | IEC application stopped because the run stop switch is on stop | IEC application stopped because the run stop switch is on stop | IEC-Anwendung wurde gestoppt, da Laufstopp-Schalter auf „Stopp“ gesetzt ist |  |  | IEC 应用程序因运行停止开关处于停止位置而停止
  Add_587202560 | Reset warm | Reset warm | Zurücksetzen (warm) |  |  | 热重置
  Add_587202561 | Reset cold | Reset cold | Zurücksetzen (kalt) |  |  | 冷重置
  Add_587202562 | Reset origin | Reset origin | Zurücksetzen (Original) |  |  | 重置原点
  Add_587202563 | Reset device | Reset device | Gerät zurücksetzen |  |  | 重置设备
  Add_637534224 | Software watchdog of IEC task expired | Software watchdog of IEC task expired | Software-Watchdog von IEC-Aufgabe abgelaufen |  |  | IEC 任务的软件看门狗已过期
  Add_637534225 | Hardware watchdog expired. Global software error | Hardware watchdog expired. Global software error | Hardware-Watchdog abgelaufen. Globaler Software-Fehler |  |  | 硬件看门狗已过期. 全局软件错误
  Add_637534226 | I/O configuration error | I/O configuration error | E/A-Konfigurationsfehler |  |  | I/O 配置错误
  Add_637534227 | Checksum error after program download | Checksum error after program download | Prüfsummenfehler nach Programm-Download |  |  | 程序下载后校验和错误
  Add_637534228 | Fieldbus error | Fieldbus error | Feldbus-Fehler |  |  | Fieldbus 错误
  Add_637534229 | I/O update error | I/O update error | E/A-Update-Fehler |  |  | I/O 更新错误
  Add_637534230 | Cycle time exceeded | Cycle time exceeded | Zykluszeit überschritten |  |  | 已超出循环时间
  Add_637534231 | Program too large for online change | Program too large for online change | Programm zu groß für Online-Änderung |  |  | 程序过大，无法在线更改
  Add_637534232 | Unresolved external references | Unresolved external references | Nicht aufgelöste externe Referenzen |  |  | 未解决的外部引用
  Add_637534233 | Download was rejected | Download was rejected | Download abgelehnt |  |  | 下载被拒绝
  Add_637534234 | Boot project not loaded because retain variables could not be relocated | Boot project not loaded because retain variables could not be relocated | Boot-Projekt nicht geladen, da Retain-Variablen nicht geladen werden konnten |  |  | 由于保留变量无法重定位，引导项目未加载
  Add_637534235 | Boot project not loaded and deleted | Boot project not loaded and deleted | Boot-Projekt nicht geladen und gelöscht |  |  | 引导项目未加载且已删除
  Add_637534236 | Out of heap memory | Out of heap memory | Kein Heap-Speicher mehr verfügbar |  |  | 堆内存不足
  Add_637534237 | Retain memory corrupt or cannot be mapped | Retain memory corrupt or cannot be mapped | Retain-Speicher beschädigt oder kann nicht zugeordnet werden |  |  | 保留内存损坏或无法映射
  Add_637534238 | Boot project could be loaded but caused an exception | Boot project could be loaded but caused an exception | Boot-Projekt konnte aufgrund einer Ausnahme nicht geladen werden |  |  | 引导项目可以加载，但会导致异常
  Add_637534241 | Target of the boot project doesn't match the current target | Target of the boot project doesn't match the current target | Ziel von Boot-Projekt stimmt nicht mit aktuellem Ziel überein |  |  | 引导项目的目标与当前目标不匹配
  Add_637534242 | Error at scheduling IEC tasks | Error at scheduling IEC tasks | Fehler bei der Zeitplanung von IEC-Aufgaben |  |  | 安排 IEC 任务时出错
  Add_637534243 | Checksum of downloaded file does not match | Checksum of downloaded file does not match | Diskrepanz bei Prüfsumme der heruntergeladenen Datei |  |  | 下载文件的校验和不匹配
  Add_637534244 | Retain identity does not match to current boot application program identity | Retain identity does not match to current boot application program identity | Retain-Identität stimmt nicht mit aktueller Identität des Boot-Anwendungsprogramms überein |  |  | 保留标识与当前引导应用程序标识不匹配
  Add_637534245 | IEC task configuration failed | IEC task configuration failed | IEC-Aufgabenkonfiguration fehlgeschlagen |  |  | IEC 任务配置失败
  Add_637534246 | Application is running on wrong target. Can be used for library protection! | Application is running on wrong target. Can be used for library protection! | Anwendung läuft über falsches Ziel. Kann zum Schutz der Bibliothek verwendet werden! |  |  | 应用程序在错误的目标上运行. 可用于库保护！
  Add_637534288 | Illegal instruction | Illegal instruction | Ungültige Anweisung |  |  | 非法指令
  Add_637534289 | Access violation | Access violation | Zugriffsverletzung |  |  | 访问冲突
  Add_637534290 | Privileged instruction | Privileged instruction | Privilegierte Anweisung |  |  | 特权指令
  Add_637534292 | Stack overflow | Stack overflow | Stack-Überlauf |  |  | 堆栈溢出
  Add_637534293 | Invalid disposition | Invalid disposition | Ungültige Löschung |  |  | 处置无效
  Add_637534294 | Invalid handle | Invalid handle | Ungültiger Handle |  |  | 句柄无效
  Add_637534295 | Guard page | Guard page | Guard-Seite |  |  | 守护页面
  Add_637534296 | Double fault | Double fault | Doppelfehler |  |  | 双重故障
  Add_637534297 | Invalid OpCode | Invalid OpCode | Ungültiger OpCode |  |  | 操作码无效
  Add_637534464 | Data type misalignment | Data type misalignment | Abweichender Datentyp |  |  | 数据类型不一致
  Add_637534465 | Array bounds exceeded | Array bounds exceeded | Array-Grenzen überschritten |  |  | 超出数组边界
  Add_637534466 | Division by zero | Division by zero | Division durch Null |  |  | 除以零
  Add_637534467 | Overflow | Overflow | Überlauf |  |  | 溢出
  Add_637534468 | Non continuable | Non continuable | Nicht fortführbar |  |  | 非连续性
  Add_637534469 | Processor load watchdog of all IEC tasks detected | Processor load watchdog of all IEC tasks detected | Prozessorlast-Watchdog aller IEC-Aufgaben erkannt |  |  | 检测到所有 IEC 任务的处理器负载看门狗
  Add_637534544 | FPU: Unspecified error | FPU: Unspecified error | FPU: Nicht spezifizierter Fehler |  |  | FPU：不明错误
  Add_637534545 | FPU: Denormalized operand | FPU: Denormalized operand | FPU: Denormalisierter Operand |  |  | FPU：非规范化操作数
  Add_637534546 | FPU: Division by zero | FPU: Division by zero | FPU: Division durch Null |  |  | FPU：除以零
  Add_637534547 | FPU: Inexact result | FPU: Inexact result | FPU: Ungenaues Ergebnis |  |  | FPU：结果不准确
  Add_637534548 | FPU: Invalid operation | FPU: Invalid operation | FPU: Ungültige Operation |  |  | FPU：无效操作
  Add_637534549 | FPU: Overflow | FPU: Overflow | FPU: Überlauf |  |  | FPU：溢出
  Add_637534550 | FPU: Stack check | FPU: Stack check | FPU: Stack-Prüfung |  |  | FPU：堆栈检查
  Add_637534551 | FPU: Underflow | FPU: Underflow | FPU: Unterlauf |  |  | FPU：下溢
  Add_637534720 | Hardware breakpoint | Hardware breakpoint | Hardware-Breakpoint |  |  | 硬件断点
  Add_637538320 | Omitted cycle watchdog | Omitted cycle watchdog | Zyklus-Watchdog ausgelassen |  |  | 已省略循环看门狗
  Err_10 | Medium has almost used its complete spare capacity or is already dead, action required | Medium has almost used its complete spare capacity or is already dead, action required | Fast die gesamte freie Kapazität des Mediums ist belegt oder es ist bereits deaktiviert, Maßnahme erforderlich |  |  | 介质的全部备用容量已经接近用尽或已经用尽，需要采取措施
  Err_11 | Type scaling on PLC startup failed | Type scaling on PLC startup failed | Typskalierung bei SPS-Start fehlgeschlagen |  |  | PLC 启动时的类型扩展失败
  Err_12 | Flash is temporary protected (read only) | Flash is temporary protected (read only) | Flash-Speicher ist temporär geschützt (schreibgeschützt) |  |  | 闪存受到临时保护（只读）
  Err_17 | Error setting parameters | Error setting parameters | Fehlereinstellungsparameter |  |  | 设置参数时出错
  Err_18 | At least one not found | At least one not found | Mindestens eine/r/s nicht gefunden |  |  | 至少有一个未找到
  Err_19 | Unable to read at least one value | Unable to read at least one value | Lesen von mindestens einem Fehler fehlgeschlagen |  |  | 无法读取至少一个值
  Err_2 | Resource failure | Resource failure | Ressourcenfehler |  |  | 资源故障
  Err_20 | Invalid value of "Error LED" | Invalid value of "Error LED" | Ungültiger Wert für „Fehler-LED“ |  |  | “错误 LED”的值无效
  Err_21 | Invalid value of "Check battery" | Invalid value of "Check battery" | Ungültiger Wert für „Überwachung Batteriestatus“ |  |  | “检查电池”的值无效
  Err_22 | Error at initialization | Error at initialization | Fehler bei der Initialisierung |  |  | 初始化时出错
  Err_23 | Wrong version of firmware | Wrong version of firmware | Falsche Firmware-Version |  |  | 固件版本错误
  Err_24 | Invalid value of parameter "Diagnosis, stop on error class" | Invalid value of parameter "Diagnosis, stop on error class" | Ungültiger Wert für Parameter „Diagnose, Stopp bei Fehlerklasse“ |  |  | 参数“诊断，出现错误类别时停止”的值无效
  Err_25 | Invalid value of parameter "Diagnosis, add Plc name to node name" | Invalid value of parameter "Diagnosis, add Plc name to node name" | Ungültiger Wert für Parameter „Diagnose, SPS-Namen zum Knotennamen hinzufügen“ |  |  | 参数“诊断，将 PLC 名称添加到节点名称”的值无效
  Err_26 | Invalid value of parameter "Reboot at powerfail" | Invalid value of parameter "Reboot at powerfail" | Ungültiger Wert für Parameter „Bei Stromausfall neu starten“ |  |  | 参数“电源故障时重新引导”的值无效
  Err_27 | Failed to set parameter "Reboot at powerfail" | Failed to set parameter "Reboot at powerfail" | Einstellen von Parameter „Bei Stromausfall neu starten“ fehlgeschlagen |  |  | 无法设置参数“电源故障时重新引导”
  Err_28 | Value of parameter "Missed Cycle Task behaviour" is not in range | Value of parameter "Missed Cycle Task behaviour" is not in range | Wert von Parameter „Verhalten bei versäumter Zyklusaufgabe“ liegt außerhalb des zulässigen Bereichs |  |  | 参数“错过周期任务行为”的值不在范围内
  Err_29 | Combination of plugged option boards is invalid | Combination of plugged option boards is invalid | Kombination von eingesteckten Optionskarten ist ungültig |  |  | 插入的选项板组合无效
  Err_3 | Timeout | Timeout | Timeout |  |  | 超时
  Err_30 | Value of parameter "Priority Scheme" is not in range | Value of parameter "Priority Scheme" is not in range | Wert von Parameter „Prioritätsschema“ liegt außerhalb des zulässigen Bereichs |  |  | 参数“优先级方案”的值不在范围内
  Err_31 | PLC did not go to RUN mode due to an active error, whose severity exceeds value of parameter 'stop on error class' | PLC did not go to RUN mode due to an active error, whose severity exceeds value of parameter 'stop on error class' | SPS ist aufgrund eines aktiven Fehlers, dessen Schweregrad den Wert für Parameter „Stoppen bei Fehlerklasse“ überschreitet, nicht in den RUN-Modus gewechselt |  |  | 由于存在严重程度超出“出错时停止类”参数值的活动错误，PLC 未进入运行模式。
  Err_32 | PLC went to STOP mode due to occurence of an error, whose severity exceeds value of parameter 'stop on error class' | PLC went to STOP mode due to occurence of an error, whose severity exceeds value of parameter 'stop on error class' | SPS ist aufgrund eines Fehlers, dessen Schweregrad den Wert für Parameter „Stoppen bei Fehlerklasse“ überschreitet, in den STOPP-Modus gewechselt |  |  | 由于发生严重程度超出“出错时停止类”参数值的错误，PLC 进入停止模式。
  Err_33 | PLC went to RUN mode | PLC went to RUN mode | SPS in RUN-Modus gewechselt |  |  | PLC 进入运行模式
  Err_34 | PLC went to STOP mode | PLC went to STOP mode | SPS in STOPP-Modus gewechselt |  |  | PLC 进入停止模式
  Err_35 | IEC application has been reset | IEC application has been reset | IEC-Anwendung wurde zurückgesetzt |  |  | IEC 应用程序已重置
  Err_36 | Online change of IEC application has been performed | Online change of IEC application has been performed | Online-Änderung von IEC-Anwendung wurde vorgenommen |  |  | 已执行 IEC 应用程序的在线更改
  Err_37 | Full download of an IEC application has been performed | Full download of an IEC application has been performed | Vollständiger Download einer IEC-Anwendung wurde ausgeführt |  |  | 已执行 IEC 应用程序的完整下载
  Err_38 | IEC application caused an exception | IEC application caused an exception | IEC-Anwendung hat eine Ausnahme verursacht |  |  | IEC 应用程序导致异常
  Err_39 | PLC did not go to RUN mode since reboot has to be performed first | PLC did not go to RUN mode since reboot has to be performed first | SPS ist nicht in den RUN-Modus gewechselt, da zunächst Neustart ausgeführt werden musste |  |  | PLC 未进入运行模式，必须先执行重新引导
  Err_40 | Value of parameter "Reboot on E2" is not in range | Value of parameter "Reboot on E2" is not in range | Wert von Parameter „Neu starten bei E2“ liegt außerhalb des zulässigen Bereichs |  |  | 参数“在 E2 时重新引导”的值不在范围内
  Err_41 | PLC went to reboot due to occurence of an E2 error | PLC went to reboot due to occurence of an E2 error | SPS ist aufgrund eines E2-Fehlers neu gestartet |  |  | 由于发生 E2 错误，PLC 重新引导
  Err_42 | No boot project loaded | No boot project loaded | Kein Boot-Projekt geladen |  |  | 引导项目未加载
  Err_43 | Boot project loaded | Boot project loaded | Boot-Projekt geladen |  |  | 引导项目已加载
  Err_44 | Loading boot project failed due to failing load of retain data | Loading boot project failed due to failing load of retain data | Laden von Boot-Projekt aufgrund von Fehler beim Laden von Retain-Daten fehlgeschlagen |  |  | 由于保留数据加载失败，引导项目加载失败
  Err_45 | Loading boot project failed due to mismatch of retain data | Loading boot project failed due to mismatch of retain data | Laden von Boot-Projekt aufgrund einer Diskrepanz der Retain-Daten fehlgeschlagen |  |  | 由于保留数据不匹配，引导项目加载失败
  Err_46 | Loading boot project failed due to insufficient license for application | Loading boot project failed due to insufficient license for application | Laden von Boot-Projekt aufgrund einer unzureichenden Anwendungslizenz fehlgeschlagen |  |  | 由于应用程序许可证不足，引导项目加载失败
  Err_47 | Loading boot project failed due to unspecified reason | Loading boot project failed due to unspecified reason | Laden von Boot-Projekt aus unbekanntem Grund fehlgeschlagen |  |  | 由于不明原因，引导项目加载失败
  Err_48 | Backup failed | Backup failed | Backup fehlgeschlagen |  |  | 备份失败
  Err_49 | Restore failed | Restore failed | Wiederherstellung fehlgeschlagen |  |  | 还原失败
  Err_50 | Invalid value of parameter "Enable diagnosis history" | Invalid value of parameter "Enable diagnosis history" | Ungültiger Wert für Parameter „Diagnosehistorie aktivieren“ |  |  | 参数“启用诊断历史记录”的值无效
  Err_51 | Invalid value of parameter "Maximum number of entries in diagnosis history" | Invalid value of parameter "Maximum number of entries in diagnosis history" | Ungültiger Wert für Parameter „Maximale Anzahl von Einträgen in Diagnosehistorie“ |  |  | 参数“诊断历史记录中的最大条目数”的值无效
  Err_52 | Invalid value of parameter "Maximum size of extended diagnosis data in diagnosis history" | Invalid value of parameter "Maximum size of extended diagnosis data in diagnosis history" | Ungültiger Wert für Parameter „Maximale Größe von erweiterten Diagnosedaten in Diagnosehistorie“ |  |  | 参数“诊断历史记录中扩展诊断数据的最大大小”的值无效
  Err_53 | System partition free space has fallen below pre-warn threshold -> Please contact your ABB representative to fix this issue | System partition free space has fallen below pre-warn threshold -> Please contact your ABB representative to fix this issue | Freier Speicherplatz der Systempartition ist unter Vorwarngrenze gesunken -> Zur Behebung dieses Problems entsprechenden ABB-Vertreter kontaktieren |  |  | 系统分区可用空间已降至低于预警阈值 -> 请联系您的 ABB 代表以解决此问题
  Err_54 | System Partition has run out of space -> Please contact your ABB representative to fix this issue and replace the CPU as soon as possible | System Partition has run out of space -> Please contact your ABB representative to fix this issue and replace the CPU as soon as possible | Systempartition hat keinen Speicherplatz mehr -> Zur Behebung dieses Problems entsprechenden ABB-Vertreter kontaktieren und schnellstmöglich CPU austauschen |  |  | 系统分区空间已用尽 -> 请联系您的 ABB 代表以解决此问题，并且尽快更换 CPU
  Err_55 | IEC project prevented from going to RUN mode, see PLC log for details | IEC project prevented from going to RUN mode, see PLC log for details |  |  |  | 
  Err_8 | Empty or missing | Empty or missing | Leer oder fehlt |  |  | 空或缺失
  Err_9 | Medium has used 80% of its spare capacity | Medium has used 80% of its spare capacity | 80 % der freien Kapazität von Medium belegt |  |  | 介质的备用容量已经使用 80%
  Hwd_0 | CPU | CPU | CPU |  |  | CPU
  Sub1_0 | CPU | CPU | CPU |  |  | CPU
  Sub1_14 | I/O bus | I/O bus | E/A-Bus |  |  | I/O 总线
  Sub1_19 | Flashdisk | Flashdisk | Flashdisk |  |  | 闪盘
  Sub1_21 | Display | Display | Anzeige |  |  | 显示
  Sub1_22 | Battery | Battery | Batterie |  |  | 电池
  Sub2_0 | Device | Device | Gerät |  |  | 设备
  Sub2_2 | Parameter | Parameter | Parameter |  |  | 参数
  Sub2_5 | Index | Index | Index |  |  | 索引
  Sub2_6 | Application | Application | Anwendung |  |  | 应用程序
  Sub2_7 | Bootproject | Bootproject |  |  |  | 
  Sub2_8 | Component | Component |  |  |  | 
  Sub4_1 | too big | too big | zu groß |  |  | 过大
  Sub4_2 | too small | too small | zu klein |  |  | 过小
  Sub4_3 | unequal | unequal | ungleich |  |  | 不等于
  Sub4_4 | equal | equal | gleich |  |  | 等于 *)
